FUNCTION EqualsPoint2D : BOOL
VAR_INPUT
	p1 : Point2D;
	p2 : Point2D;
	epsilon : Point2D;
END_VAR

EqualsPoint2D := EqualsLREAL(p1.X, p2.X, epsilon.X)
			AND EqualsLREAL(p1.Y, p2.Y, epsilon.Y);

END_FUNCTION

(* stored: Version 1.1.0.1
   POU EqualsPoint2D: Id {cfbe5c7c-4031-081c-3d4b-77d3c4948084}, SpecialFunc None *)
